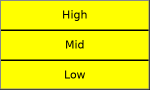
VISUALIZATION Floor  // 150x90
VAR_INPUT
	LS_Floor :ST_LevelSensors;
END_VAR
    Rectangle (0,60 150x30), "Low", colour toggle: LS_Floor.Low
    Rectangle (0,30 150x30), "Mid", colour toggle: LS_Floor.Mid
    Rectangle (0,0 150x30), "High", colour toggle: LS_Floor.High
END_VISUALIZATION

(* stored: Version 1.1.0.1, ProductVersion 3.1.4024.11
   Visu Floor: Id {89f159cf-c69e-417a-a2d8-477593762889} *)
